// TIA Portal V17 export
// export: Created 2025-04-05T09:21:23.2412683Z, ExportSetting WithDefaults, DisplayName Totally Integrated Automation Portal, DisplayVersion V17, DisplayName TIA Portal Openness, DisplayVersion V17, DisplayName TIA Portal Version Control Interface, DisplayVersion V17, DisplayName STEP 7 Professional, DisplayVersion V17, DisplayName STEP 7 Safety, DisplayVersion V17, DisplayName WinCC Advanced, DisplayVersion V17
FUNCTION_BLOCK "Foutca"   // FB1, GRAPH
VERSION : 0.1
// stored: AcknowledgeErrorsRequired true, AutoNumber true, GraphVersion 6.0, InitialValuesAcquisition false, IsIECCheckEnabled false, LanguageInNetworks LAD, LockOperatingMode false, PermanentILProcessingInMANMode false, SetENOAutomatically false, SkipSteps false, UDAEnableTagReadback false, WithAlarmHandling true
   // inherited from GRAPH_BASE
   VAR
      OFF_SQ_BASE : Bool;
   END_VAR
   VAR_INPUT
      OFF_SQ { ExternalAccessible := 'False'; ExternalVisible := 'False'; ExternalWritable := 'False'} : Bool := false;   // Turn sequence off
      INIT_SQ { ExternalAccessible := 'False'; ExternalVisible := 'False'; ExternalWritable := 'False'} : Bool := false;   // Set sequence to initial state
      ACK_EF { ExternalAccessible := 'False'; ExternalVisible := 'False'; ExternalWritable := 'False'} : Bool := false;   // Acknowledge all errors and faults
      S_PREV { ExternalAccessible := 'False'; ExternalVisible := 'False'; ExternalWritable := 'False'} : Bool := false;   // Output previous step in parameter S_NO
      S_NEXT { ExternalAccessible := 'False'; ExternalVisible := 'False'; ExternalWritable := 'False'} : Bool := false;   // Indicate next step in parameter S_NO
      SW_AUTO { ExternalAccessible := 'False'; ExternalVisible := 'False'; ExternalWritable := 'False'} : Bool := false;   // Automatic mode
      SW_TAP { ExternalAccessible := 'False'; ExternalVisible := 'False'; ExternalWritable := 'False'} : Bool := false;   // Semiautomatic/switch with transition
      SW_TOP { ExternalAccessible := 'False'; ExternalVisible := 'False'; ExternalWritable := 'False'} : Bool := false;   // Semiautomatic/ignore transition
      SW_MAN { ExternalAccessible := 'False'; ExternalVisible := 'False'; ExternalWritable := 'False'} : Bool := false;   // Manual mode
      S_SEL { ExternalAccessible := 'False'; ExternalVisible := 'False'; ExternalWritable := 'False'} : Int := 0;   // Select step to be output to S_NO
      S_ON { ExternalAccessible := 'False'; ExternalVisible := 'False'; ExternalWritable := 'False'} : Bool := false;   // Activate step indicated in S_NO
      S_OFF { ExternalAccessible := 'False'; ExternalVisible := 'False'; ExternalWritable := 'False'} : Bool := false;   // Deactivate step indicated S_NO
      T_PUSH { ExternalAccessible := 'False'; ExternalVisible := 'False'; ExternalWritable := 'False'} : Bool := false;   // Enable transition to switch in semi automatic mode
   END_VAR
   VAR_OUTPUT
      S_NO { ExternalAccessible := 'False'; ExternalVisible := 'False'; ExternalWritable := 'False'} : Int := 0;   // Step number
      S_MORE { ExternalAccessible := 'False'; ExternalVisible := 'False'; ExternalWritable := 'False'} : Bool := false;   // More steps are available and can be shown in S_NO
      S_ACTIVE { ExternalAccessible := 'False'; ExternalVisible := 'False'; ExternalWritable := 'False'} : Bool := false;   // Step indicated in S_NO is active
      ERR_FLT { ExternalAccessible := 'False'; ExternalVisible := 'False'; ExternalWritable := 'False'} : Bool := false;   // Interlock or supervision group error
      AUTO_ON { ExternalAccessible := 'False'; ExternalVisible := 'False'; ExternalWritable := 'False'} : Bool := false;   // Automatic mode is active
      TAP_ON { ExternalAccessible := 'False'; ExternalVisible := 'False'; ExternalWritable := 'False'} : Bool := false;   // Semiautomatic mode/step with transition enabled
      TOP_ON { ExternalAccessible := 'False'; ExternalVisible := 'False'; ExternalWritable := 'False'} : Bool := false;   // Semiautomatic mode/ignore transition enabled
      MAN_ON { ExternalAccessible := 'False'; ExternalVisible := 'False'; ExternalWritable := 'False'} : Bool := false;   // Manual mode is active
   END_VAR
BEGIN
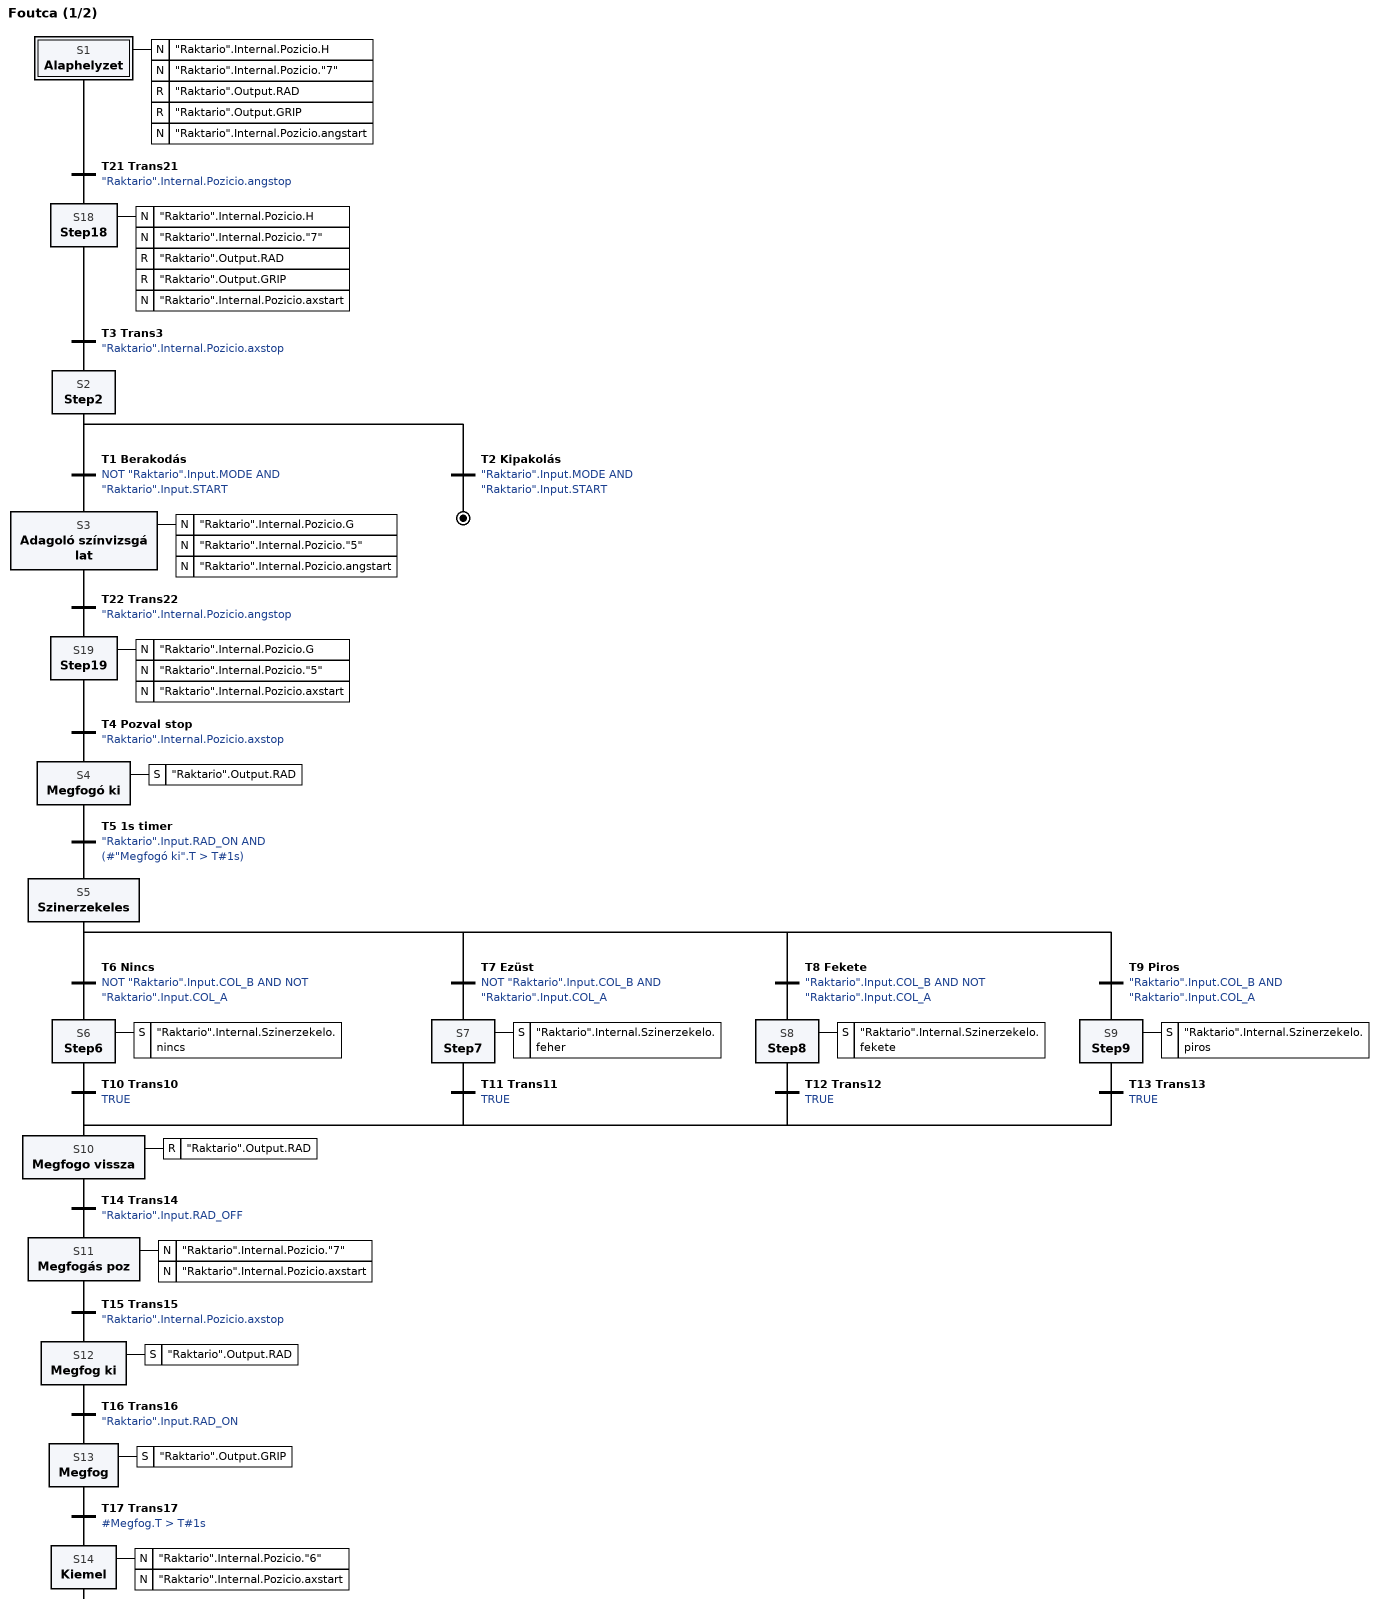
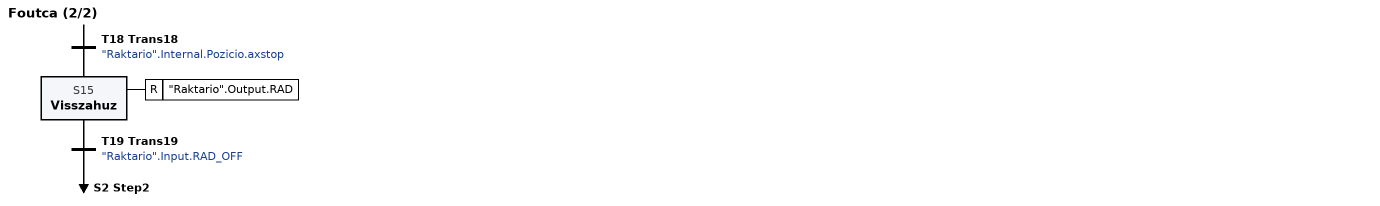
   // sequencer 1
   INITIAL_STEP Alaphelyzet:   // S1, max time T#10S, warning time T#7S
              N    "Raktario".Internal.Pozicio.H
              N    "Raktario".Internal.Pozicio."7"
              R    "Raktario".Output.RAD
              R    "Raktario".Output.GRIP
              N    "Raktario".Internal.Pozicio.angstart
   END_STEP
   TRANSITION Trans21 FROM Alaphelyzet TO Step18   // T21
      := "Raktario".Internal.Pozicio.angstop;
   END_TRANSITION
   STEP Step2:   // S2, max time T#10S, warning time T#7S
   END_STEP
   TRANSITION Berakodás FROM Step2 TO "Adagoló színvizsgálat"   // T1
      := NOT "Raktario".Input.MODE AND "Raktario".Input.START;
   END_TRANSITION
   TRANSITION Kipakolás FROM Step2 TO END   // T2
      := "Raktario".Input.MODE AND "Raktario".Input.START;
   END_TRANSITION
   STEP "Adagoló színvizsgálat":   // S3, max time T#10S, warning time T#7S
              N    "Raktario".Internal.Pozicio.G
              N    "Raktario".Internal.Pozicio."5"
              N    "Raktario".Internal.Pozicio.angstart
   END_STEP
   TRANSITION Trans22 FROM "Adagoló színvizsgálat" TO Step19   // T22
      := "Raktario".Internal.Pozicio.angstop;
   END_TRANSITION
   STEP "Megfogó ki":   // S4, max time T#10S, warning time T#7S
              S    "Raktario".Output.RAD
   END_STEP
   TRANSITION "1s timer" FROM "Megfogó ki" TO Szinerzekeles   // T5
      := "Raktario".Input.RAD_ON AND (#"Megfogó ki".T > T#1s);
   END_TRANSITION
   STEP Szinerzekeles:   // S5, max time T#10S, warning time T#7S
   END_STEP
   TRANSITION Nincs FROM Szinerzekeles TO Step6   // T6
      := NOT "Raktario".Input.COL_B AND NOT "Raktario".Input.COL_A;
   END_TRANSITION
   TRANSITION Ezüst FROM Szinerzekeles TO Step7   // T7
      := NOT "Raktario".Input.COL_B AND "Raktario".Input.COL_A;
   END_TRANSITION
   TRANSITION Fekete FROM Szinerzekeles TO Step8   // T8
      := "Raktario".Input.COL_B AND NOT "Raktario".Input.COL_A;
   END_TRANSITION
   TRANSITION Piros FROM Szinerzekeles TO Step9   // T9
      := "Raktario".Input.COL_B AND "Raktario".Input.COL_A;
   END_TRANSITION
   STEP Step6:   // S6, max time T#10S, warning time T#7S
              S    "Raktario".Internal.Szinerzekelo.nincs
   END_STEP
   TRANSITION Trans10 FROM Step6 TO "Megfogo vissza"   // T10
      := TRUE;
   END_TRANSITION
   STEP Step7:   // S7, max time T#10S, warning time T#7S
              S    "Raktario".Internal.Szinerzekelo.feher
   END_STEP
   TRANSITION Trans11 FROM Step7 TO "Megfogo vissza"   // T11
      := TRUE;
   END_TRANSITION
   STEP Step8:   // S8, max time T#10S, warning time T#7S
              S    "Raktario".Internal.Szinerzekelo.fekete
   END_STEP
   TRANSITION Trans12 FROM Step8 TO "Megfogo vissza"   // T12
      := TRUE;
   END_TRANSITION
   STEP Step9:   // S9, max time T#10S, warning time T#7S
              S    "Raktario".Internal.Szinerzekelo.piros
   END_STEP
   TRANSITION Trans13 FROM Step9 TO "Megfogo vissza"   // T13
      := TRUE;
   END_TRANSITION
   STEP "Megfogo vissza":   // S10, max time T#10S, warning time T#7S
              R    "Raktario".Output.RAD
   END_STEP
   TRANSITION Trans14 FROM "Megfogo vissza" TO "Megfogás poz"   // T14
      := "Raktario".Input.RAD_OFF;
   END_TRANSITION
   STEP "Megfogás poz":   // S11, max time T#10S, warning time T#7S
              N    "Raktario".Internal.Pozicio."7"
              N    "Raktario".Internal.Pozicio.axstart
   END_STEP
   TRANSITION Trans15 FROM "Megfogás poz" TO "Megfog ki"   // T15
      := "Raktario".Internal.Pozicio.axstop;
   END_TRANSITION
   STEP "Megfog ki":   // S12, max time T#10S, warning time T#7S
              S    "Raktario".Output.RAD
   END_STEP
   TRANSITION Trans16 FROM "Megfog ki" TO Megfog   // T16
      := "Raktario".Input.RAD_ON;
   END_TRANSITION
   STEP Megfog:   // S13, max time T#10S, warning time T#7S
              S    "Raktario".Output.GRIP
   END_STEP
   TRANSITION Trans17 FROM Megfog TO Kiemel   // T17
      := #Megfog.T > T#1s;
   END_TRANSITION
   STEP Kiemel:   // S14, max time T#10S, warning time T#7S
              N    "Raktario".Internal.Pozicio."6"
              N    "Raktario".Internal.Pozicio.axstart
   END_STEP
   TRANSITION Trans18 FROM Kiemel TO Visszahuz   // T18
      := "Raktario".Internal.Pozicio.axstop;
   END_TRANSITION
   STEP Visszahuz:   // S15, max time T#10S, warning time T#7S
              R    "Raktario".Output.RAD
   END_STEP
   TRANSITION Trans19 FROM Visszahuz TO Step2   // T19, jump
      := "Raktario".Input.RAD_OFF;
   END_TRANSITION
   STEP Step18:   // S18, max time T#10S, warning time T#7S
              N    "Raktario".Internal.Pozicio.H
              N    "Raktario".Internal.Pozicio."7"
              R    "Raktario".Output.RAD
              R    "Raktario".Output.GRIP
              N    "Raktario".Internal.Pozicio.axstart
   END_STEP
   TRANSITION Trans3 FROM Step18 TO Step2   // T3
      := "Raktario".Internal.Pozicio.axstop;
   END_TRANSITION
   STEP Step19:   // S19, max time T#10S, warning time T#7S
              N    "Raktario".Internal.Pozicio.G
              N    "Raktario".Internal.Pozicio."5"
              N    "Raktario".Internal.Pozicio.axstart
   END_STEP
   TRANSITION "Pozval stop" FROM Step19 TO "Megfogó ki"   // T4
      := "Raktario".Internal.Pozicio.axstop;
   END_TRANSITION
END_FUNCTION_BLOCK
